Fanuc KAREL source: kt00605.KL

-- PROVISIONAL review KL for V1013-1; original PC SHA256 27c270e959d066b1d8298856982cc21dd8dedbc92e723ec06b4f29f0d323cd63
-- Incomplete behavior may be omitted. Consult companion uncertainty JSON. Do not deploy.
PROGRAM KT00605
%NOLOCKGROUP
VAR
  I1 : INTEGER
  I2 : INTEGER
  OUT : REAL
BEGIN
  -- UNRESOLVED_PC offsets 5-16; opcodes 2E,23
  -- UNRESOLVED_PC offsets 21-32; opcodes 2E,23
  -- UNRESOLVED_PC offsets 37-48; opcodes 2E,23
  -- UNRESOLVED_PC offsets 53-64; opcodes 2E,23
  -- UNRESOLVED_PC offsets 69-83; opcodes 21,51,64,23
  -- UNRESOLVED_PC offsets 88-92; opcodes 7F
END KT00605
